// TIA Portal project "3M-8" (V16)

(* hardware
DEVICE "S7-1200 station_1"  S7-1200 Station
   slot 0: "Rack_0"  S7-1200 Rack  Rack  V1.0
   slot 1: "PLC_1"  CPU 1212C AC/DC/Rly  6ES7 212-1BE40-0XB0  V4.0
*)

// ===== PLC "PLC_1"  CPU 1212C AC/DC/Rly =====

VAR_GLOBAL   // PLC tag table "Default tag table"
   ""start1"" AT %I0.2 : Bool;
   ""stop1"" AT %I0.4 : Bool;
   ""start2"" AT %I0.3 : Bool;
   ""K1"" AT %Q0.0 : Bool;
   ""k2"" AT %Q0.1 : Bool;
   ""K3"" AT %Q0.2 : Bool;
END_VAR